// TIA Portal V20 export
FUNCTION_BLOCK "FB_LoaderAxis"   // FB206, SCL
{ S7_Optimized_Access := 'TRUE' }
// stored: AutoNumber false, MemoryReserve 100, SetENOAutomatically false
   VAR_INPUT
      iPLCModeReq : Bool;   // Axis Managed by PLC Request
      iCNCModeReq : Bool;   // Axis Managed by CNC Request
      iU1StartReq : Bool;   // Axis U1 Start Request
      iU2StartReq : Bool;   // Axis U2 Start Request
      iVStartReq : Bool;   // Axis V Start Request
      iWStartReq : Bool;   // Axis W Start Request
      iU1PosSetPoint : Real;   // Axis U1 Position Setpoint
      iU2PosSetPoint : Real;   // Axis U2 Position Setpoint
      iVPosSetPoint : Real;   // Axis V Position Setpoint
      iWPosSetPoint : Real;   // Axis W Position Setpoint
   END_VAR
   VAR_OUTPUT
      oU1InPos : Bool;   // Axis U1 Position Reached
      oU2InPos : Bool;   // Axis U2 Position Reached
      oVInPos : Bool;   // Axis V Position Reached
      oWInPos : Bool;   // Axis W Position Reached
   END_VAR
   VAR
      sAxisPLCMode : Bool := false;
      sAxisCNCMode : Bool := false;
      sAllAxisPLCMode : Bool := false;
      sAllAxisCNCMode : Bool := false;
      sU1StartMove : Bool;
      sU2StartMove : Bool;
      sVStartMove : Bool;
      sWStartMove : Bool;
      sU1MoveError : Bool;
      sU2MoveError : Bool;
      sVMoveError : Bool;
      sWMoveError : Bool;
      sU1InPos : Bool;
      sU2InPos : Bool;
      sVInPos : Bool;
      sWInPos : Bool;
      sU1SetPos : Real;
      sU2SetPos : Real;
      sVSetPos : Real;
      sWSetPos : Real;
      sU1MoveState : Byte;
      sU2MoveState : Byte;
      sVMoveState : Byte;
      sWMoveState : Byte;
      sU1ActFeedRate : LReal;
      sU2ActFeedRate : LReal;
      sVActFeedRate : LReal;
      sWActFeedRate : LReal;
      sU1DrivedByPLC : Bool;
      sU2DrivedByPLC : Bool;
      sVDrivedByPLC : Bool;
      sWDrivedByPLC : Bool;
      sU1Positioning { ExternalAccessible := 'False'; ExternalVisible := 'False'; ExternalWritable := 'False'} : Bool;
      sU2Positioning { ExternalAccessible := 'False'; ExternalVisible := 'False'; ExternalWritable := 'False'} : Bool;
      sVPositioning { ExternalAccessible := 'False'; ExternalVisible := 'False'; ExternalWritable := 'False'} : Bool;
      sWPositioning { ExternalAccessible := 'False'; ExternalVisible := 'False'; ExternalWritable := 'False'} : Bool;
      sFeedActive : Bool;
   END_VAR
BEGIN
   REGION Update Inputs
       #sU1StartMove := #iU1StartReq;
       #sU2StartMove := #iU2StartReq;
       #sVStartMove  := #iVStartReq;
       #sWStartMove  := #iWStartReq;

       #sU1SetPos := #iU1PosSetPoint;
       #sU2SetPos := #iU2PosSetPoint;
       #sVSetPos  := #iVPosSetPoint;
       #sWSetPos  := #iWPosSetPoint;
   END_REGION


   REGION Feed Active/Axis moving
       #sU1Positioning := "LBP_Axis05_U1".E_PosAxis AND "LBP_Axis05_U1".E_PLCASp;
       #sU2Positioning := "LBP_Axis06_U2".E_PosAxis AND "LBP_Axis06_U2".E_PLCASp;
       #sVPositioning  := "LBP_Axis07_V".E_PosAxis  AND "LBP_Axis07_V".E_PLCASp;
       #sWPositioning  := "LBP_Axis08_W".E_PosAxis  AND "LBP_Axis08_W".E_PLCASp;

       #sFeedActive := //  A least 1 axis is moving
       ("LBP_Chan1".A_FD_OR <> B#16#1)  // Speed more than 0
       AND (#sU1Positioning             // Axis06 U1 moving
           OR #sU2Positioning           // Axis09 U2 moving
           OR #sVPositioning            // Axis07 V  moving
           OR #sWPositioning);          // Axis08 W  moving
   END_REGION

   REGION Axis CNC mode (Only when NC in JOG Mode)
       IF #sAxisPLCMode
           AND #iCNCModeReq
           OR "MCP1_In".reset
           OR NOT "DB_DataFromSafety".EmergencyStop THEN
           #sAxisCNCMode := TRUE;
           #sAxisPLCMode := FALSE;
       END_IF;

       #sAllAxisCNCMode :=
           NOT "LBP_Axis05_U1".E_PLCASp
       AND NOT "LBP_Axis06_U2".E_PLCASp
       AND NOT "LBP_Axis07_V".E_PLCASp
       AND NOT "LBP_Axis08_W".E_PLCASp;
   END_REGION

   REGION Axis PLC mode (When NC Not in JOG Mode)
       IF #sAxisCNCMode
            AND #iPLCModeReq THEN
           #sAxisPLCMode := TRUE;
           #sAxisCNCMode := FALSE;
       END_IF;

       #sAllAxisPLCMode :=
           "LBP_Axis05_U1".E_PLCASp
       AND "LBP_Axis06_U2".E_PLCASp
       AND "LBP_Axis07_V".E_PLCASp
       AND "LBP_Axis08_W".E_PLCASp;
   END_REGION

   REGION Set axis feed rate
       #sU1ActFeedRate := "DB_AxisPosition".sAxis05_U1."$MA_MAX_AX_VELO";
       #sU2ActFeedRate := "DB_AxisPosition".sAxis06_U2."$MA_MAX_AX_VELO";
       #sVActFeedRate := "DB_AxisPosition".sAxis07_V."$MA_MAX_AX_VELO";
       IF (("DB_LoaderShuttle1".sIntLoadUnload.sCurrent_Step_NB = 100
           OR "DB_LoaderShuttle1".sIntLoadUnload.sCurrent_Step_NB = 110)
           AND "DB_AxisPosition".sAxis08_W."$AA_IM" <= "DB_AxisPosMachinePLC".Axis_W.Shuttle_1.Approach)

           OR (("DB_LoaderShuttle2".sIntLoadUnload.sCurrent_Step_NB = 100
           OR "DB_LoaderShuttle2".sIntLoadUnload.sCurrent_Step_NB = 110)
           AND "DB_AxisPosition".sAxis08_W."$AA_IM" <= "DB_AxisPosMachinePLC".Axis_W.Shuttle_2.Approach)

           OR (("DB_LoaderShuttle1".sIntLoadUnloadOP.sCurrent_Step_NB = 100
           OR "DB_LoaderShuttle1".sIntLoadUnloadOP.sCurrent_Step_NB = 110)
           AND "DB_AxisPosition".sAxis08_W."$AA_IM" <= "DB_AxisPosMachinePLC".Axis_W.Shuttle_1.Approach)

           OR (("DB_LoaderShuttle2".sIntLoadUnloadOP.sCurrent_Step_NB = 100
           OR "DB_LoaderShuttle2".sIntLoadUnloadOP.sCurrent_Step_NB = 110)
           AND "DB_AxisPosition".sAxis08_W."$AA_IM" <= "DB_AxisPosMachinePLC".Axis_W.Shuttle_2.Approach)

           OR (("DB_LoaderShuttle1".sIntLoadUnloadOP.sCurrent_Step_NB = 190
           OR "DB_LoaderShuttle1".sIntLoadUnloadOP.sCurrent_Step_NB = 200)
           AND "DB_AxisPosition".sAxis08_W."$AA_IM" <= "DB_AxisPosMachinePLC".Axis_W.Shuttle_1.Approach)

           OR (("DB_LoaderShuttle2".sIntLoadUnloadOP.sCurrent_Step_NB = 190
           OR "DB_LoaderShuttle2".sIntLoadUnloadOP.sCurrent_Step_NB = 200)
           AND "DB_AxisPosition".sAxis08_W."$AA_IM" <= "DB_AxisPosMachinePLC".Axis_W.Shuttle_2.Approach)

           OR(("DB_LoaderFixture".sFixtureLoading.sCurrent_Step_NB = 80
           OR "DB_LoaderFixture".sFixtureLoading.sCurrent_Step_NB = 85)
           AND "DB_AxisPosition".sAxis08_W."$AA_IM" <= "DB_AxisPosMachinePLC".Axis_W.Fixture.Approach)


       THEN
           #sWActFeedRate := "DB_AxisPosition".sAxis08_W."$MA_JOG_VELO";
       ELSE
           #sWActFeedRate := "DB_AxisPosition".sAxis08_W."$MA_MAX_AX_VELO";
       END_IF;
   END_REGION

   REGION Check axis drived by PLC
       // Axis U1
       #sU1DrivedByPLC := "LBP_Axis05_U1".E_RefSyn1
       AND #sAxisPLCMode
       AND NOT #sAxisCNCMode;

       // Axis U2
       #sU2DrivedByPLC := "LBP_Axis06_U2".E_RefSyn1
       AND #sAxisPLCMode
       AND NOT #sAxisCNCMode;

       // Axis V
       #sVDrivedByPLC := "LBP_Axis07_V".E_RefSyn1
       AND #sAxisPLCMode
       AND NOT #sAxisCNCMode;

       // Axis W
       #sWDrivedByPLC := "LBP_Axis08_W".E_RefSyn1
       AND #sAxisPLCMode
       AND NOT #sAxisCNCMode;
   END_REGION

   REGION Set axis PLC/CNC mode
       // Axis U1 (Always drived by PLC in Auto Mode)
       "LBP_Axis05_U1".A_NCASpStrobe := #sU1DrivedByPLC
       AND NOT "LBP_Axis05_U1".E_PLCASp
       OR NOT #sU1DrivedByPLC
       AND "LBP_Axis05_U1".E_PLCASp;

       "LBP_Axis05_U1".A_PLCASp := #sU1DrivedByPLC;

       // Axis U2 (Always drived by PLC in Auto Mode)
       "LBP_Axis06_U2".A_NCASpStrobe := #sU2DrivedByPLC
       AND NOT "LBP_Axis06_U2".E_PLCASp
       OR NOT #sU2DrivedByPLC
       AND "LBP_Axis06_U2".E_PLCASp;

       "LBP_Axis06_U2".A_PLCASp := #sU2DrivedByPLC;

       // Axis V (Always drived by PLC in Auto Mode)
       "LBP_Axis07_V".A_NCASpStrobe := #sVDrivedByPLC
       AND NOT "LBP_Axis07_V".E_PLCASp
       OR NOT #sVDrivedByPLC
       AND "LBP_Axis07_V".E_PLCASp;

       "LBP_Axis07_V".A_PLCASp := #sVDrivedByPLC;

       // Axis W (Always drived by PLC in Auto Mode)
       "LBP_Axis08_W".A_NCASpStrobe := #sWDrivedByPLC
       AND NOT "LBP_Axis08_W".E_PLCASp
       OR NOT #sWDrivedByPLC
       AND "LBP_Axis08_W".E_PLCASp;

       "LBP_Axis08_W".A_PLCASp := #sWDrivedByPLC;
   END_REGION

   REGION Delete distance to go
       // Axis U1
       "LBP_Axis05_U1".A_DelDTGSpReset := NOT #sU1StartMove
       AND "LBP_Axis05_U1".E_PLCASp
       OR "MCP1_In".reset
       OR "LBP_ModeGroup".E_REF;

       // Axis U2
       "LBP_Axis06_U2".A_DelDTGSpReset := NOT #sU2StartMove
       AND "LBP_Axis06_U2".E_PLCASp
       OR "MCP1_In".reset
       OR "LBP_ModeGroup".E_REF;

       // Axis V
       "LBP_Axis07_V".A_DelDTGSpReset := NOT #sVStartMove
       AND "LBP_Axis07_V".E_PLCASp
       OR "MCP1_In".reset
       OR "LBP_ModeGroup".E_REF;

       // Axis W
       "LBP_Axis08_W".A_DelDTGSpReset := NOT #sWStartMove
       AND "LBP_Axis08_W".E_PLCASp
       OR "MCP1_In".reset
       OR "LBP_ModeGroup".E_REF;
   END_REGION

   REGION Axis positioning
       // Axis U1
       "LBP_CtrlAxisSpindle"(Start := #sU1StartMove AND #sU1DrivedByPLC,
                             Stop := FALSE,
                             Funct := B#16#5,
                             Mode := B#16#0,
                             AxisNo := 5,
                             Pos := #sU1SetPos,
                             FRate := LREAL_TO_REAL(#sU1ActFeedRate),
                             InPos => #sU1InPos,
                             Error => #sU1MoveError,
                             State => #sU1MoveState);

       IF #sU1InPos
           OR "MCP1_In".reset
           OR #sU1MoveError THEN
           #sU1StartMove := FALSE;
       END_IF;

       IF #sU1MoveError THEN
           "LBP_AlarmMsgs".UserA[08].A70UUxx[08] := TRUE;
       END_IF;

       // Axis U2
       "LBP_CtrlAxisSpindle"(Start := #sU2StartMove AND #sU2DrivedByPLC,
                             Stop := FALSE,
                             Funct := B#16#5,
                             Mode := B#16#0,
                             AxisNo := 6,
                             Pos := #sU2SetPos,
                             FRate := LREAL_TO_REAL(#sU2ActFeedRate),
                             InPos => #sU2InPos,
                             Error => #sU2MoveError,
                             State => #sU2MoveState);
       IF #sU2MoveState <> 0 THEN
           "DB_WAF".U2States := #sU2MoveState;
       END_IF;

       IF #sU2InPos
           OR "MCP1_In".reset
           OR #sU2MoveError THEN
           #sU2StartMove := FALSE;
       END_IF;

       IF #sU2MoveError THEN
           "LBP_AlarmMsgs".UserA[08].A70UUxx[09] := TRUE;
       END_IF;

       // Axis V
       "LBP_CtrlAxisSpindle"(Start := #sVStartMove AND #sVDrivedByPLC,
                             Stop := FALSE,
                             Funct := B#16#5,
                             Mode := B#16#0,
                             AxisNo := 7,
                             Pos := #sVSetPos,
                             FRate := LREAL_TO_REAL(#sVActFeedRate),
                             InPos => #sVInPos,
                             Error => #sVMoveError,
                             State => #sVMoveState);

       IF #sVInPos
           OR "MCP1_In".reset
           OR #sVMoveError THEN
           #sVStartMove := FALSE;
       END_IF;

       IF #sVMoveError THEN
           "LBP_AlarmMsgs".UserA[08].A70UUxx[10] := TRUE;
       END_IF;

       // Axis W
       "LBP_CtrlAxisSpindle"(Start := #sWStartMove AND #sWDrivedByPLC,
                             Stop := FALSE,
                             Funct := B#16#5,
                             Mode := B#16#0,
                             AxisNo := 8,
                             Pos := #sWSetPos,
                             FRate := LREAL_TO_REAL(#sWActFeedRate),
                             InPos => #sWInPos,
                             Error => #sWMoveError,
                             State => #sWMoveState);

       IF #sWInPos
           OR "MCP1_In".reset
           OR #sWMoveError THEN
           #sWStartMove := FALSE;
       END_IF;

       IF #sWMoveError THEN
           "LBP_AlarmMsgs".UserA[08].A70UUxx[11] := TRUE;
       END_IF;
   END_REGION

   REGION Update Outputs
       #oU1InPos := #sU1InPos;
       #oU2InPos := #sU2InPos;
       #oVInPos  := #sVInPos;
       #oWInPos  := #sWInPos;
   END_REGION
END_FUNCTION_BLOCK
